// TIA Portal V19 export
VAR_GLOBAL   // PLC tag table "A03_302"
   A0302_SpintoreLongitudinale_Ls_Minimo AT %I269.1 : Bool;   // 1602SQ1
   A0302_SpintoreLongitudinale_Ls_Massimo AT %I269.2 : Bool;   // 1602SQ2
   A0302_SpintoreLongitudinale_Verticale_Ls_Rest_1 AT %I269.3 : Bool;   // 1610SQ1
   A0302_SpintoreLongitudinale_Verticale_Ls_Work_1 AT %I269.4 : Bool;   // 1610SQ2
   A0302_SpintoreLongitudinale_Orizzontale_Ls_Rest_2 AT %I269.5 : Bool;   // 1610SQ3
   A0302_SpintoreLongitudinale_Orizzontale_Ls_Work_2 AT %I269.6 : Bool;   // 1610SQ4
   A0302_SpintoreLongitudinale_Orizzontale_V_Rest_1 AT %Q273.4 : Bool;   // 1610YV1
   A0302_SpintoreLongitudinale_Orizzontale_V_Work_1 AT %Q273.5 : Bool;   // 1610YV2
   A0302_SpintoreLongitudinale_Orizzontale_V_Rest_2 AT %Q273.6 : Bool;   // 1610YV3
   A0302_SpintoreLongitudinale_Orizzontale_V_Work_2 AT %Q273.7 : Bool;   // 1610YV4
   A0302_SpintoreLongitudinale_PezzoEstratto_Phc AT %I269.7 : Bool;   // 1614BF1
   A0302_Bordatrice_ControlloConnettoreBanco_4_Lato_1 AT %I270.0 : Bool;   // 1830X1A
   A0302_Bordatrice_Banco_4_Lato_1_Phc_AtEntry AT %I270.1 : Bool;   // 1833SQ1
   A0302_Bordatrice_Banco_4_Lato_1_Phc_AtExit AT %I270.2 : Bool;   // 1833SQ2
   "A0302_Bordatrice_Spalla_4.1_Ls_Minimo" AT %I270.3 : Bool;   // 1842SQ1
   "A0302_Bordatrice_Spalla_4.1_Ls_Massimo" AT %I270.4 : Bool;   // 1842SQ2
   "A0302_Bordatrice_Spalla_4.3_Motore_Apre" AT %Q6.0 : Bool;   // 1850KM1
   "A0302_Bordatrice_Spalla_4.3_Motore_Chiude" AT %Q6.1 : Bool;   // 1850KM2
   "A0302_Bordatrice_Spalla_4.3_Motore_AnomaliaTermica" AT %I5.5 : Bool;   // 1850QF1
   "A0302_Bordatrice_Spalla_4.3_Ls_AperturaMinima" AT %I270.5 : Bool;   // 1851SQ1
   "A0302_Bordatrice_Spalla_4.3_Ls_AperturaMassima" AT %I270.6 : Bool;   // 1851SQ2
   "A0302_Bordatrice_Spalla_4.5_Motore_Apre" AT %Q6.2 : Bool;   // 1855KM1
   "A0302_Bordatrice_Spalla_4.5_Motore_Chiude" AT %Q6.3 : Bool;   // 1855KM2
   "A0302_Bordatrice_Spalla_4.5_Motore_AnomaliaTermica" AT %I5.6 : Bool;   // 1855QF1
   "A0302_Bordatrice_Spalla_4.5_Ls_AperturaMinima" AT %I270.7 : Bool;   // 1856SQ1
   "A0302_Bordatrice_Spalla_4.5_Ls_AperturaMassima" AT %I271.0 : Bool;   // 1856SQ2
   "A0302_Bordatrice_Spalla_4.7_Motore_Apre" AT %Q6.4 : Bool;   // 1860KM1
   "A0302_Bordatrice_Spalla_4.7_Motore_Chiude" AT %Q6.5 : Bool;   // 1860KM2
   "A0302_Bordatrice_Spalla_4.7_Motore_AnomaliaTermica" AT %I5.7 : Bool;   // 1860QF1
   "A0302_Bordatrice_Spalla_4.7_Ls_AperturaMinima" AT %I271.1 : Bool;   // 1861SQ1
   "A0302_Bordatrice_Spalla_4.7_Ls_AperturaMassima" AT %I271.2 : Bool;   // 1861SQ2
   "A0302_Bordatrice_Spalla_4.9_Motore_Apre" AT %Q6.6 : Bool;   // 1865KM1
   "A0302_Bordatrice_Spalla_4.9_Motore_Chiude" AT %Q6.7 : Bool;   // 1865KM2
   "A0302_Bordatrice_Spalla_4.9_Motore_AnomaliaTermica" AT %I6.0 : Bool;   // 1865QF1
   "A0302_Bordatrice_Spalla_4.9_Ls_AperturaMinima" AT %I271.3 : Bool;   // 1866SQ1
   "A0302_Bordatrice_Spalla_4.9_Ls_AperturaMassima" AT %I271.4 : Bool;   // 1866SQ2
   A0302_Bordatrice_ControlloConnettoreBanco_4_Lato_2 AT %I271.5 : Bool;   // 1880X1A
   A0302_Bordatrice_Banco_4_Lato_2_Phc_AtEntry AT %I271.6 : Bool;   // 1883SQ1
   A0302_Bordatrice_Banco_4_Lato_2_PhcPhc_AtExit AT %I271.7 : Bool;   // 1883SQ2
   "A0302_Bordatrice_Spalla_4.2_Ls_Minimo" AT %I272.0 : Bool;   // 1892SQ1
   "A0302_Bordatrice_Spalla_4.2_Ls_Massimo" AT %I272.1 : Bool;   // 1892SQ2
   "A0302_Bordatrice_Spalla_4.4_Motore_Apre" AT %Q7.0 : Bool;   // 1900KM1
   "A0302_Bordatrice_Spalla_4.4_Motore_Chiude" AT %Q7.1 : Bool;   // 1900KM2
   "A0302_Bordatrice_Spalla_4.4_Motore_AnomaliaTermica" AT %I6.1 : Bool;   // 1900QF1
   "A0302_Bordatrice_Spalla_4.4_Ls_Minimo" AT %I272.2 : Bool;   // 1901SQ1
   "A0302_Bordatrice_Spalla_4.4_Ls_Massimo" AT %I272.3 : Bool;   // 1901SQ2
   "A0302_Bordatrice_Spalla_4.6_Motore_Apre" AT %Q7.2 : Bool;   // 1905KM1
   "A0302_Bordatrice_Spalla_4.6_Motore_Chiude" AT %Q7.3 : Bool;   // 1905KM2
   "A0302_Bordatrice_Spalla_4.6_Motore_AnomaliaTermica" AT %I6.2 : Bool;   // 1905QF1
   "A0302_Bordatrice_Spalla_4.6_Ls_Minimo" AT %I272.4 : Bool;   // 1906SQ1
   "A0302_Bordatrice_Spalla_4.6_Ls_Massimo" AT %I272.5 : Bool;   // 1906SQ2
   "A0302_Bordatrice_Spalla_4.8_Motore_Apre" AT %Q7.4 : Bool;   // 1910KM1
   "A0302_Bordatrice_Spalla_4.8_Motore_Chiude" AT %Q7.5 : Bool;   // 1910KM2
   "A0302_Bordatrice_Spalla_4.8_Motore_AnomaliaTermica" AT %I6.3 : Bool;   // 1910QF1
   "A0302_Bordatrice_Spalla_4.8_Ls_Minimo" AT %I272.6 : Bool;   // 1911SQ1
   "A0302_Bordatrice_Spalla_4.8_Ls_Massimo" AT %I272.7 : Bool;   // 1911SQ2
   "A0302_Bordatrice_Spalla_4.10_Motore_Apre" AT %Q7.6 : Bool;   // 1915KM1
   "A0302_Bordatrice_Spalla_4.10_Motore_Chiude" AT %Q7.7 : Bool;   // 1915KM2
   "A0302_Bordatrice_Spalla_4.10_Motore_AnomaliaTermica" AT %I6.4 : Bool;   // 1915QF1
   "A0302_Bordatrice_Spalla_4.10_Ls_Minimo" AT %I273.0 : Bool;   // 1916SQ1
   "A0302_Bordatrice_Spalla_4.10_Ls_Massimo" AT %I273.1 : Bool;   // 1916SQ2
   A0302_Bordatrice_Lubrificazione_LivelloMinimo AT %I273.2 : Bool;   // 1960SL1
   A0302_Bordatrice_V_Lubrificazione AT %Q274.0 : Bool;   // 1960YV1
   A0302_HU_Cytropack_Ready AT %I302.2 : Bool;   // 1970
   A0302_HU_Cytropack_Enable AT %Q302.3 : Bool;   // 1970
   A0302_HU_Cytropack_FaultReset AT %Q302.4 : Bool;   // 1970
   A0302_HU_Cytropack_Warning AT %I302.3 : Bool;   // 1970
   A0302_HU_Cytropack_SetBit0 AT %Q302.5 : Bool;   // 1970
   A0302_HU_Cytropack_SetBit1 AT %Q302.6 : Bool;   // 1970
   A0302_HU_Cytropack_AlimentazioneGruppoChiller AT %Q2.2 : Bool;   // 1975KM1
   A0302_HU_Cytropack_Chiller_Ok AT %I302.4 : Bool;   // 1975KM1
   A0302_HU_Cytropack_Chiller_Start AT %Q302.7 : Bool;   // 1975KA1
   A0302_Rulliera_Lato_1_Testa_Phc_PezzoRallentamentoBattuta AT %I352.0 : Bool;   // 2010BF2
   A0302_Rulliera_Lato_1_Testa_Phc_PezzoStopBattuta AT %I352.1 : Bool;   // 2010BF3
   A0302_Rulliera_Lato_2_Coda_Phc_PezzoInArrivo AT %I302.5 : Bool;   // 2012BF1
   A0302_Rulliera_Lato_2_Coda_Phc_PezzoDopoBattuta AT %I302.6 : Bool;   // 2012BF2
   A0302_Rulliera_Lato_2_Coda_Phc_1_ControlloNuovoPezzo AT %I302.7 : Bool;   // 2012BF3
   A0302_Rulliera_Lato_2_Coda_Phc_2_ControlloNuovoPezzo AT %I303.0 : Bool;   // 2012BF4
   A0302_Rulliera_Lato_2_Coda_Phc_3_ControlloNuovoPezzo AT %I303.1 : Bool;   // 2012BF5
   A0302_Centratori_Centraggio_1_Coda_Ls_Basso AT %I303.2 : Bool;   // 2020SQ1
   A0302_Centratori_Centraggio_1_Coda_Ls_Alto AT %I303.3 : Bool;   // 2020SQ2
   A0302_Centratori_Centraggio_1_Coda_Ls_Aperto AT %I303.4 : Bool;   // 2020SQ3
   A0302_Centratori_Centraggio_1_Coda_Ls_Chiuso AT %I303.5 : Bool;   // 2020SQ4
   A0302_Centratori_Centraggio_1_Coda_V_Basso AT %Q310.0 : Bool;   // 2020YV1
   A0302_Centratori_Centraggio_1_Coda_V_Alto AT %Q310.1 : Bool;   // 2020YV2
   A0302_Centratori_Centraggio_1_Coda_V_Aperto AT %Q310.2 : Bool;   // 2020YV3
   A0302_Centratori_Centraggio_1_Coda_V_Chiuso AT %Q310.3 : Bool;   // 2020YV4
   A0302_PezziAccumolo_Scivolo_2_Phc_1 AT %I353.2 : Bool;   // 2060SQ1
   A0302_PezziAccumolo_Scivolo_2_Phc_2 AT %I353.3 : Bool;   // 2060SQ2
   A0302_Ax_Pareggiatore_Testa_Ls_Minimo AT %I353.6 : Bool;   // 2102SQ1
   A0302_Ax_Pareggiatore_Testa_Ls_Massimo AT %I353.7 : Bool;   // 2102SQ2
   A0302_Ax_Pareggiatore_Testa_AntiCollisione AT %I354.0 : Bool;   // 2102SQ3
   A0302_Pareggiatore_Testa_Bloccaggio_V_Rest AT %Q352.1 : Bool;   // 2110YV1
   A0302_Pareggiatore_Testa_Bloccaggio_V_Work AT %Q352.2 : Bool;   // 2110YV2
   A0302_Pareggiatore_Testa_Bloccaggio_LatoMotore_Ls_Rest AT %I354.1 : Bool;   // 2110SQ1
   A0302_Pareggiatore_Testa_Bloccaggio_LatoOperatore_Ls_Rest AT %I354.2 : Bool;   // 2110SQ2
   A0302_Pareggiatore_Testa_Bloccaggio_LatoMotore_Ls_Work AT %I354.3 : Bool;   // 2110SQ3
   A0302_Pareggiatore_Testa_Bloccaggio_LatoOperatore_Ls_Work AT %I354.4 : Bool;   // 2110SQ4
   A0302_Manipolatore_Ax_Testa_Ls_Minimo AT %I355.1 : Bool;   // 2142SQ1
   A0302_Manipolatore_Ax_Testa_Ls_Massimo AT %I355.2 : Bool;   // 2142SQ2
   A0302_Manipolatore_Testa_Ls_Alto AT %I355.3 : Bool;   // 2150SQ1
   A0302_Manipolatore_Testa_Ls_Basso AT %I355.4 : Bool;   // 2150SQ2
   A0302_Manipolatore_Testa_Magnete_Ls_Rest AT %I355.5 : Bool;   // 2150SQ3
   A0302_Manipolatore_Testa_Magnete_Ls_Work AT %I355.6 : Bool;   // 2150SQ4
   A0302_Manipolatore_Testa_V_Alto AT %Q361.4 : Bool;   // 2150YV1
   A0302_Manipolatore_Testa_V_Basso AT %Q361.5 : Bool;   // 2150YV2
   A0302_Manipolatore_Testa_V_Rest AT %Q361.6 : Bool;   // 2150YV3
   A0302_Manipolatore_Testa_V_Work AT %Q361.7 : Bool;   // 2150YV4
   A0302_Carrello_Testa_V_Rest AT %Q362.0 : Bool;   // 2151YV1
   A0302_Carrello_Testa_V_Work AT %Q362.1 : Bool;   // 2151YV2
   A0302_Ax_Pareggiatore_Coda_Ls_Minimo AT %I303.6 : Bool;   // 2182SQ1
   A0302_Ax_Pareggiatore_Coda_Ls_Massimo AT %I303.7 : Bool;   // 2182SQ2
   A0302_Ax_Pareggiatore_Coda_AntiCollisione AT %I304.0 : Bool;   // 2182SQ3
   A0302_Pareggiatore_Coda_Bloccaggio_V_Rest AT %Q303.0 : Bool;   // 2190YV1
   A0302_Pareggiatore_Coda_Bloccaggio_V_Work AT %Q303.1 : Bool;   // 2190YV2
   A0302_Pareggiatore_Coda_Bloccaggio_LatoMotore_Ls_Rest AT %I304.1 : Bool;   // 2190SQ1
   A0302_Pareggiatore_Coda_Bloccaggio_LatoOperatore_Ls_Rest AT %I304.2 : Bool;   // 2190SQ2
   A0302_Pareggiatore_Coda_Bloccaggio_LatoMotore_Ls_Work AT %I304.3 : Bool;   // 2190SQ3
   A0302_Pareggiatore_Coda_Bloccaggio_LatoOperatore_Ls_Work AT %I304.4 : Bool;   // 2190SQ4
   A0302_Pareggiatore_Coda_Centraggio_Ls_Alto AT %I304.5 : Bool;   // 2200SQ1
   A0302_Pareggiatore_Coda_Centraggio_Ls_Basso AT %I304.6 : Bool;   // 2200SQ2
   A0302_Pareggiatore_Coda_Centraggio_V_Alto AT %Q310.4 : Bool;   // 2200YV1
   A0302_Pareggiatore_Coda_Centraggio_V_Basso AT %Q310.5 : Bool;   // 2200YV2
   A0302_Pareggiatore_Coda_Longitudinale_V_Aperto AT %Q303.2 : Bool;   // 2202YV1
   A0302_Pareggiatore_Coda_Longitudinale_V_Chiuso AT %Q303.3 : Bool;   // 2202YV2
   A0302_Pareggiatore_Coda_Longitudinale_Ls_Aperto AT %I304.7 : Bool;   // 2202SQ1
   A0302_Pareggiatore_Coda_Longitudinale_Ls_Chiuso AT %I305.0 : Bool;   // 2202SQ2
   A0302_Manipolatore_Ax_Coda_Ls_Minimo AT %I305.1 : Bool;   // 2222SQ1
   A0302_Manipolatore_Ax_Coda_Ls_Massimo AT %I305.2 : Bool;   // 2222SQ2
   A0302_Manipolatore_Coda_Ls_Alto AT %I305.3 : Bool;   // 2230SQ1
   A0302_Manipolatore_Coda_Ls_Basso AT %I305.4 : Bool;   // 2230SQ2
   A0302_Manipolatore_Coda_Magnete_Ls_Rest AT %I305.5 : Bool;   // 2230SQ3
   A0302_Manipolatore_Coda_Magnete_Ls_Work AT %I305.6 : Bool;   // 2230SQ4
   A0302_Manipolatore_Coda_V_Alto AT %Q310.6 : Bool;   // 2230YV1
   A0302_Manipolatore_Coda_V_Basso AT %Q310.7 : Bool;   // 2230YV2
   A0302_Manipolatore_Coda_V_Rest AT %Q311.0 : Bool;   // 2230YV3
   A0302_Manipolatore_Coda_V_Work AT %Q311.1 : Bool;   // 2230YV4
   A0302_Carrello_Coda_V_Rest_1 AT %Q311.2 : Bool;   // 2231YV1
   A0302_Carrello_Coda_V_Work_1 AT %Q311.3 : Bool;   // 2231YV2
   A0302_Carrello_Coda_V_Rest_2 AT %Q311.4 : Bool;   // 2231YV3
   A0302_Carrello_Coda_V_Work_2 AT %Q311.5 : Bool;   // 2231YV4
   A0302_AI_Ammortizatore_Posizionamento AT %IW924 : Int;   // 512A1 - 1612A1
   A0302_AI_Pareggiatore_Coda_Longitudinale_Posizionamento AT %IW932 : Int;   // 532A1 - 2204A1
   A0302_AI_Pareggiatore_Coda_Bloccaggio_Pressostato AT %IW936 : Int;   // 533A1 - 2191SB1
   A0302_AI_Pareggiatore_Testa_Bloccaggio_Pressostato AT %IW940 : Int;   // 552A1 - 2111B1
   A0302_Centraggio_Battuta_Testa_Ls_Riposo_Alto AT %I354.5 : Bool;   // 2120SQ1
   A0302_Centraggio_Battuta_Testa_Ls_Lavoro_Basso AT %I354.6 : Bool;   // 2120SQ2
   A0302_Centraggio_Battuta_Testa_Ls_Riposo_Aperto AT %I354.7 : Bool;   // 2120SQ3
   A0302_Centraggio_Battuta_Testa_Ls_Lavoro_Chiuso AT %I355.0 : Bool;   // 2120SQ4
   A0302_Pareggiatore_Testa_Centraggio_Vrt_V_WorkBasso AT %Q361.1 : Bool;   // 2120YV2
   A0302_Pareggiatore_Testa_Centraggio_Orz_V_Aperto AT %Q361.2 : Bool;   // 2120YV3
   A0302_Pareggiatore_Testa_Centraggio_Orz_V_Chiuso AT %Q361.3 : Bool;   // 2120YV4
   A0302_Pareggiatore_Testa_Centraggio_Vrt_V_RestAlto AT %Q361.0 : Bool;   // 2120YV1
END_VAR
